// TIA Portal project "TS_Stoliar_DP" (V20)

(* hardware
DEVICE "S7-1200 G2 station_1"  S7-1200 G2 Station
   slot 0: "Rack_0"  S71200G2 Rack  Rack  V1.0
   slot 1: "G2_PLC_1"  CPU 1214C DC/DC/DC  6ES7 214-1AH50-0XB0  V1.0
   slot 9: "AI2/AQ2 signal board_1"  AI2/AQ2 signal board  6ES7 233-4HD50-0XB0  V1.0
*)

// ===== PLC "G2_PLC_1"  CPU 1214C DC/DC/DC =====

VAR_GLOBAL   // PLC tag table "Default tag table"
   "VENT" AT %QW80 : Int;
   "SPIR" AT %QW82 : Int;
   "SNIMAC1" AT %IW80 : Int;
   "SNIMAC2" AT %IW82 : Int;
END_VAR

DATA_BLOCK "DATA"   // DB1
{ S7_Optimized_Access := 'TRUE' }
VERSION : 0.1
   VAR
      block_enable : Bool;
      y1 : Real;
      y2 : Real;
      u : Real;
      vent : Real;
      "time" : LReal;
      ypb : Real;
      u_pb : Real;
   END_VAR
BEGIN
END_DATA_BLOCK

DATA_BLOCK "Current_time_DB"   // DB2
{ S7_Optimized_Access := 'TRUE' }
VERSION : 0.1
// stored: InstanceOfName Current_time
"Current_time"
BEGIN
END_DATA_BLOCK

DATA_BLOCK "PREP"   // DB3
{ S7_Optimized_Access := 'TRUE' }
VERSION : 0.1
   VAR
      r_l : Real;
      r_g : Real;
      r_gf : Real;
      u_g : Real;
      u_l : Real;
      active_g : Bool;
      Ki_l : Real;
      Kp_l : Real;
   END_VAR
BEGIN
END_DATA_BLOCK

DATA_BLOCK "FB_PI_TS05_DB"   // DB5
{ S7_Optimized_Access := 'TRUE' }
VERSION : 0.1
// stored: InstanceOfName FB_PI_TS05
"FB_PI_TS05"
BEGIN
END_DATA_BLOCK

DATA_BLOCK "FB_PI_LOGGER_DB"   // DB6
{ S7_Optimized_Access := 'TRUE' }
VERSION : 0.1
// stored: InstanceOfName FB_PI_LOGGER
"FB_PI_LOGGER"
BEGIN
END_DATA_BLOCK

// folder: System blocks/Program resources

DATA_BLOCK "IEC_Timer_0_DB"   // DB4
{ S7_Optimized_Access := 'TRUE' }
AUTHOR : Simatic
FAMILY : IEC
NAME : IEC_TMR
VERSION : 1.0
// stored: InstanceOfName IEC_TIMER
"IEC_TIMER"
BEGIN
END_DATA_BLOCK

// folder: (top level)

FUNCTION_BLOCK "FB_PI_TS05"   // FB1, SCL
{ S7_Optimized_Access := 'TRUE' }
VERSION : 0.1
   VAR_INPUT
      Y : Real;
      Setpoint_pb : Real;
      Enable : Bool;
   END_VAR
   VAR_OUTPUT
      U : Real;
      Ypb : Real;
      vent : Real;
   END_VAR
   VAR
      Integrator : Real;
   END_VAR
   VAR_TEMP
      "E" : Real;
      DU : Real;
   END_VAR
   VAR CONSTANT
      Kp : Real := 3.58;
      Ki : Real := 1.84;
      Ts : Real := 0.1;
      U_pb : Real := 4.0;
      DU_min : Real := -4.0;
      DU_max : Real := 6.0;
   END_VAR
BEGIN
   IF NOT #Enable THEN
       #U := #U_pb;
       #DU := 0.0;
       #E := 0.0;
       #Integrator := 0.0;
       #Ypb := #Y;
       #vent := 6.0;

   ELSE
       #E := #Setpoint_pb - (#Y - #Ypb);
       #Integrator := #Integrator + #E * #Ts;

       #DU := #Kp * #E + #Ki * #Integrator;

       IF #DU > #DU_max THEN
           #DU := #DU_max;
       ELSIF #DU < #DU_min THEN
           #DU := #DU_min;
       END_IF;

       #U := #U_pb + #DU;
       #vent := 6.0;
   END_IF;
END_FUNCTION_BLOCK

FUNCTION_BLOCK "FB_PI_LOGGER"   // FB2, SCL
{ S7_Optimized_Access := 'TRUE' }
VERSION : 0.1
   VAR_INPUT
      CurrentTimeSec : LReal;
      u : Real;
      y : Real;
      r : Real;
      ypb : Real;
      Enable : Bool;
   END_VAR
   VAR_OUTPUT
      SampleCount : DInt;
      Full : Bool;
   END_VAR
   VAR
      idx : DInt;
      TimeLog_s : Array[0..9999] of LReal;
      ULOG : Array[0..9999] of Real;
      YLOG : Array[0..9999] of Real;
      RLOG : Array[0..9999] of Real;
      YPBLOG : Array[0..9999] of Real;
   END_VAR
BEGIN
   IF NOT #Full AND #Enable THEN
       IF #idx <= 9999 THEN
           #TimeLog_s[#idx] := #CurrentTimeSec;
           #ULOG[#idx] := #u;
           #YLOG[#idx] := #y;
           #RLOG[#idx] := #r;
           #YPBLOG[#idx] := #ypb;

           #idx := #idx + 1;
           #SampleCount := #idx;
       ELSE
           #Full := TRUE;
       END_IF;
   END_IF;
END_FUNCTION_BLOCK

FUNCTION_BLOCK "Current_time"   // FB3, SCL
{ S7_Optimized_Access := 'TRUE' }
VERSION : 0.1
   VAR_OUTPUT
      CurrentTimeSec : LReal;
   END_VAR
   VAR
      started : Bool;
      retVal : Int;
      startTime : DTL;
      currentTime : DTL;
      elapsedTime : Time;
   END_VAR
BEGIN
   #retVal := RD_SYS_T(OUT => #currentTime);

   IF (NOT #started) AND (#retVal = 0) THEN
       #startTime := #currentTime;
       #started := TRUE;
   END_IF;

   IF #started AND (#retVal = 0) THEN
       #elapsedTime := T_DIFF(IN1 := #currentTime, IN2 := #startTime);
       #CurrentTimeSec := DINT_TO_LREAL(TIME_TO_DINT(#elapsedTime)) / 1000.0;
   ELSE
       #CurrentTimeSec := 0.0;
   END_IF;
END_FUNCTION_BLOCK

FUNCTION_BLOCK "FB_PREP_TS05"   // FB4, SCL
{ S7_Optimized_Access := 'TRUE' }
VERSION : 0.1
   VAR_INPUT
      Y : Real;
      R_g : Real;
      R_l : Real;
      Enable : Bool;
      Vent_in : Real;
   END_VAR
   VAR_OUTPUT
      U : Real;
      R_gf : Real;
      Y_pb_out : Real;
      U_pb_out : Real;
      U_g : Real;
      U_l : Real;
      Active_g : Bool;
      Kp_l_out : Real;
      Ki_l_out : Real;
      Vent_out : Real;
   END_VAR
   VAR
      X_f1 : Real;
      X_f2 : Real;
      I_l : Real;
      I_g : Real;
      Y_hist : Array[0..29] of Real;
      U_hist : Array[0..29] of Real;
      R_g_prev : Real;
      Active_g_m : Bool;
      Y_pb : Real;
      U_pb : Real;
      Initialized : Bool;
      Y_pb_table : Array[0..2] of Real;
      U_pb_table : Array[0..2] of Real;
      Kp_l_table : Array[0..2] of Real;
      Ki_l_table : Array[0..2] of Real;
   END_VAR
   VAR_TEMP
      E_l : Real;
      E_g : Real;
      U_tmp : Real;
      Lower_bound : Real;
      Upper_bound : Real;
      Y_pb_new : Real;
      U_pb_new : Real;
      Count_ok : Int;
      Idx_pb : Int;
      I : Int;
      Active_g_new : Bool;
      Active_l : Bool;
      Kp_l : Real;
      Ki_l : Real;
      Y_pb_est : Real;
      U_pb_est : Real;
      Dist_pb : Real;
      Dist_i : Real;
      X_f1_new : Real;
      X_f2_new : Real;
      Mean_y : Real;
      Mean_u : Real;
   END_VAR
   VAR CONSTANT
      Ts : Real := 0.1;
      Kp_g : Real := 4.0;
      Ki_g : Real := 0.7;
   END_VAR
BEGIN
   IF NOT #Enable THEN
       #U := 0.0;
       #R_gf := 0.0;
       #Y_pb_out := #Y_pb;
       #U_pb_out := #U_pb;
       #U_g := 0.0;
       #U_l := 0.0;
       #Active_g := #Active_g_m;
       #Kp_l_out := 0.0;
       #Ki_l_out := 0.0;
       #Vent_out := #Vent_in;
       RETURN;
   END_IF;

   // One-time initialization
   IF NOT #Initialized THEN
       #X_f1 := 0.0;
       #X_f2 := 0.0;
       #I_l := 0.0;
       #I_g := 0.0;
       #R_g_prev := #R_g;
       #Active_g_m := FALSE;
       #Y_pb := 0.0;
       #U_pb := 0.0;

       #Y_pb_table[0] := 4.4884;
       #Y_pb_table[1] := 6.3412;
       #Y_pb_table[2] := 7.7441;

       #U_pb_table[0] := 2.0;
       #U_pb_table[1] := 4.0;
       #U_pb_table[2] := 6.0;

       #Kp_l_table[0] := 2.77;
       #Kp_l_table[1] := 3.58;
       #Kp_l_table[2] := 1.83;

       #Ki_l_table[0] := 1.48;
       #Ki_l_table[1] := 1.84;
       #Ki_l_table[2] := 2.20;

       FOR #I := 0 TO 29 DO
           #Y_hist[#I] := 0.0;
           #U_hist[#I] := 0.0;
       END_FOR;

       #Initialized := TRUE;
   END_IF;

   // 1 Detect step change of global reference
   IF #R_g <> #R_g_prev THEN
       #Active_g_m := TRUE;
   END_IF;

   // 2 Filter global reference
   #R_gf := 0.01 * #X_f1;

   #X_f1_new := #X_f1 + #Ts * #X_f2;
   #X_f2_new := #X_f2 + #Ts * (-0.01 * #X_f1 - 0.2 * #X_f2 + #R_g);

   // 3 Select local operating point and PI parameters from table
   #Dist_pb := ABS(#Y_pb_table[0] - #Y_pb);
   #Idx_pb := 0;

   FOR #I := 1 TO 2 DO
       #Dist_i := ABS(#Y_pb_table[#I] - #Y_pb);
       IF #Dist_i < #Dist_pb THEN
           #Dist_pb := #Dist_i;
           #Idx_pb := #I;
       END_IF;
   END_FOR;

   #Kp_l := #Kp_l_table[#Idx_pb];
   #Ki_l := #Ki_l_table[#Idx_pb];

   // 4 Control errors
   #E_l := #R_l - (#Y - #Y_pb);
   #E_g := #R_gf - #Y;

   // 5 Control law
   IF #Active_g_m THEN
       #U_l := 0.0;
       #U_g := #Kp_g * #E_g + #Ki_g * #I_g;
   ELSE
       #U_l := #U_pb + #Kp_l * #E_l + #Ki_l * #I_l;
       #U_g := 0.0;
   END_IF;

   #U_tmp := #U_l + #U_g;

   // Saturation
   IF #U_tmp > 10.0 THEN
       #U_tmp := 10.0;
   ELSIF #U_tmp < 0.0 THEN
       #U_tmp := 0.0;
   END_IF;

   #U := #U_tmp;

   // 6 Update histories
   FOR #I := 0 TO 28 DO
       #Y_hist[#I] := #Y_hist[#I + 1];
       #U_hist[#I] := #U_hist[#I + 1];
   END_FOR;

   #Y_hist[29] := #Y;
   #U_hist[29] := #U;

   // 7 Settling detection
   #Lower_bound := #R_g - 0.03 * #R_g;
   #Upper_bound := #R_g + 0.03 * #R_g;

   #Count_ok := 0;
   FOR #I := 0 TO 29 DO
       IF (#Y_hist[#I] >= #Lower_bound) AND (#Y_hist[#I] <= #Upper_bound) THEN
           #Count_ok := #Count_ok + 1;
       END_IF;
   END_FOR;

   // Two-level switching logic
   #Y_pb_new := #Y_pb;
   #U_pb_new := #U_pb;
   #Active_g_new := #Active_g_m;

   IF #Active_g_m AND (#Count_ok >= 25) THEN
       #Mean_y := 0.0;
       #Mean_u := 0.0;

       FOR #I := 0 TO 29 DO
           #Mean_y := #Mean_y + #Y_hist[#I];
           #Mean_u := #Mean_u + #U_hist[#I];
       END_FOR;

       #Y_pb_est := #Mean_y / 30.0;
       #U_pb_est := #Mean_u / 30.0;

       #Y_pb_new := #Y_pb_est;
       #U_pb_new := #U_pb_est;
       #Active_g_new := FALSE;
   END_IF;

   IF #Active_g_m THEN
       #Active_l := FALSE;
   ELSE
       #Active_l := TRUE;
   END_IF;

   // 8 Integral states update
   IF #Active_l THEN
       #I_l := #I_l + #E_l * #Ts;
   ELSE
       #I_l := 0.0;
   END_IF;

   IF #Active_g_m THEN
       #I_g := #I_g + #E_g * #Ts;
   ELSE
       #I_g := (#U - #Kp_g * #E_g) / #Ki_g;
   END_IF;

   // 9 Memory update
   #R_g_prev := #R_g;
   #Y_pb := #Y_pb_new;
   #U_pb := #U_pb_new;
   #Active_g_m := #Active_g_new;
   #X_f1 := #X_f1_new;
   #X_f2 := #X_f2_new;

   // Outputs for monitoring/logging
   #Y_pb_out := #Y_pb;
   #U_pb_out := #U_pb;
   #Active_g := #Active_g_m;
   #Kp_l_out := #Kp_l;
   #Ki_l_out := #Ki_l;
   #Vent_out := #Vent_in;
END_FUNCTION_BLOCK

FUNCTION_BLOCK "FB_PREP_LOGGER"   // FB5, SCL
{ S7_Optimized_Access := 'TRUE' }
VERSION : 0.1
   VAR_INPUT
      t : LReal;
      r_l : Real;
      r_g : Real;
      r_gf : Real;
      y : Real;
      y_pb : Real;
      u : Real;
      u_g : Real;
      u_l : Real;
      u_pb : Real;
      active_g : Bool;
      Ki_l : Real;
      Kp_l : Real;
      Vent : Real;
   END_VAR
   VAR_OUTPUT
      SampleCount : DInt;
      Full : Bool;
   END_VAR
   VAR
      idx : DInt;
      TimeLog_s : Array[0..9999] of LReal;
      R_L_log : Array[0..9999] of Real;
      R_G_log : Array[0..9999] of Real;
      R_GF_log : Array[0..9999] of Real;
      Y_log : Array[0..9999] of Real;
      Y_PB_log : Array[0..9999] of Real;
      U_log : Array[0..9999] of Real;
      U_G_log : Array[0..9999] of Real;
      U_L_log : Array[0..9999] of Real;
      U_PB_log : Array[0..9999] of Real;
      ACTIVE_G_log : Array[0..9999] of Bool;
      KI_L_log : Array[0..9999] of Real;
      KP_L_log : Array[0..9999] of Real;
      VENT_log : Array[0..9999] of Real;
   END_VAR
BEGIN
   IF NOT #Full THEN
       IF #idx <= 9999 THEN
           #TimeLog_s[#idx] := #t;
           #R_L_log[#idx] := #r_l;
           #R_G_log[#idx] := #r_g;
           #R_GF_log[#idx] := #r_gf;
           #Y_log[#idx] := #y;
           #Y_PB_log[#idx] := #y_pb;
           #U_log[#idx] := #u;
           #U_G_log[#idx] := #u_g;
           #U_L_log[#idx] := #u_l;
           #U_PB_log[#idx] := #u_pb;
           #ACTIVE_G_log[#idx] := #active_g;
           #KI_L_log[#idx] := #Ki_l;
           #KP_L_log[#idx] := #Kp_l;
           #VENT_log[#idx] := #Vent;

           #idx := #idx + 1;
           #SampleCount := #idx;
       ELSE
           #Full := TRUE;
       END_IF;
   END_IF;
END_FUNCTION_BLOCK

FUNCTION_BLOCK "FB_PREP_SETPOINT"   // FB6, SCL
{ S7_Optimized_Access := 'TRUE' }
VERSION : 0.1
   VAR_INPUT
      t : LReal;
   END_VAR
   VAR_OUTPUT
      r_l : Real;
      r_g : Real;
   END_VAR
BEGIN
   IF #t < 1.0 THEN
       #r_g := 0.0;
   ELSIF #t < 401.0 THEN
       #r_g := 6.3412;
   ELSIF #t < 801.0 THEN
       #r_g := 4.4884;
   ELSE
       #r_g := 4.4884;
   END_IF;

   IF #t < 201.0 THEN
       #r_l := 0.0;
   ELSIF #t < 301.0 THEN
       #r_l := -0.35;
   ELSIF #t < 601.0 THEN
       #r_l := 0.0;
   ELSIF #t < 701.0 THEN
       #r_l := 0.41;
   ELSIF #t < 801.0 THEN
       #r_l := 0.0;
   ELSE
       #r_l := 0.0;
   END_IF;
END_FUNCTION_BLOCK

ORGANIZATION_BLOCK "Main"   // OB1, LAD, ProgramCycle
TITLE = "Main Program Sweep (Cycle)"
{ S7_Optimized_Access := 'TRUE' }
VERSION : 0.1
   VAR_INPUT
      Initial_Call : Bool;   // Initial call of this OB
      Remanence : Bool;   // =True, if remanent data are available
   END_VAR
   VAR_TEMP
      temp_real : Real;
   END_VAR
BEGIN

REGION Network 1
   // Time counting
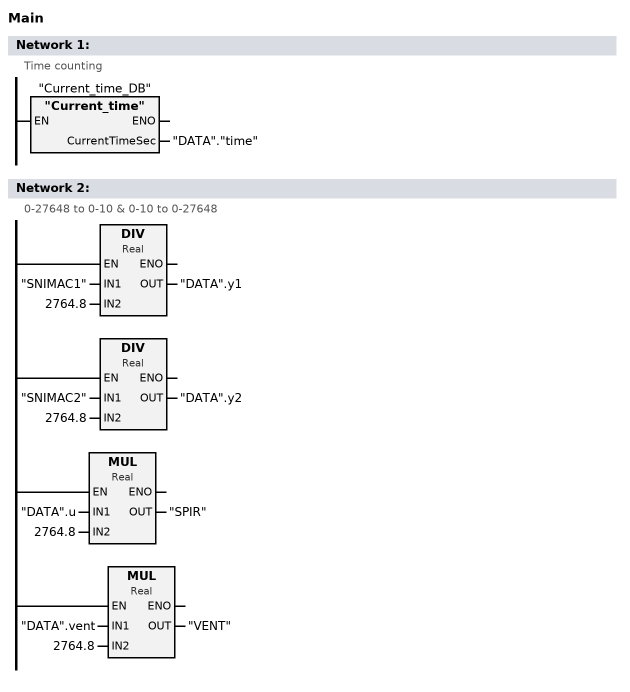
   RUNG wire#powerrail
      "Current_time_DB"(CurrentTimeSec => "DATA"."time")
   END_RUNG
   // the same network as SCL:
   "Current_time_DB"(CurrentTimeSec => "DATA"."time");   // "Current_time"
END_REGION

REGION Network 2
   // 0-27648 to 0-10 & 0-10 to 0-27648
   RUNG wire#powerrail
      { S7_Templates := "SrcType := Real" } Div(in1 := "SNIMAC1", in2 := 2764.8, out => "DATA".y1)
   END_RUNG
   RUNG wire#powerrail
      { S7_Templates := "SrcType := Real" } Div(in1 := "SNIMAC2", in2 := 2764.8, out => "DATA".y2)
   END_RUNG
   RUNG wire#powerrail
      { S7_Templates := "SrcType := Real" } Mul(in1 := "DATA".u, in2 := 2764.8, out => "SPIR")
   END_RUNG
   RUNG wire#powerrail
      { S7_Templates := "SrcType := Real" } Mul(in1 := "DATA".vent, in2 := 2764.8, out => "VENT")
   END_RUNG
   // the same network as SCL:
   "DATA".y1 := "SNIMAC1" / 2764.8;
   "DATA".y2 := "SNIMAC2" / 2764.8;
   "SPIR" := "DATA".u * 2764.8;
   "VENT" := "DATA".vent * 2764.8;
END_REGION
END_ORGANIZATION_BLOCK

ORGANIZATION_BLOCK "CyclicInterrupt"   // OB30, LAD, CyclicInterrupt
{ S7_Optimized_Access := 'TRUE' }
VERSION : 0.1
   VAR_INPUT
      Initial_Call : Bool;   // Initial call of this OB
      Event_Count : Int;   // Events discarded
   END_VAR
   VAR_TEMP   // added for the SCL form of the ladder/FBD networks
      _w1 : Bool;
   END_VAR
BEGIN

REGION Network 1
   // CONTROL LOGIC
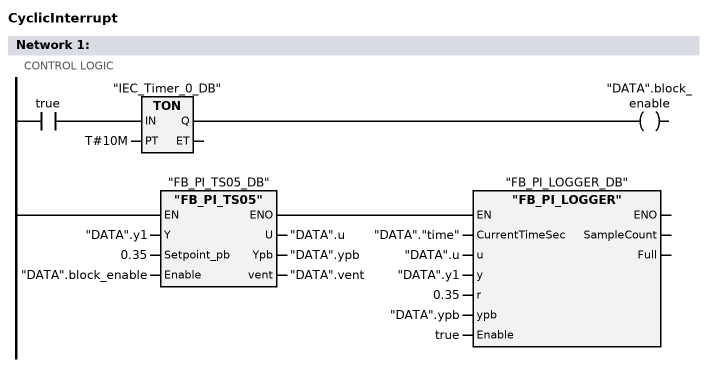
   "IEC_Timer_0_DB".TON(IN := true, PT := T#10M);
   "DATA".block_enable := "IEC_Timer_0_DB".Q;
   "FB_PI_TS05_DB"(Y := "DATA".y1,   // "FB_PI_TS05"
                   Setpoint_pb := 0.35,
                   Enable := "DATA".block_enable,
                   U => "DATA".u,
                   Ypb => "DATA".ypb,
                   vent => "DATA".vent,
                   ENO => #_w1);
   IF #_w1 THEN
       "FB_PI_LOGGER_DB"(CurrentTimeSec := "DATA"."time",   // "FB_PI_LOGGER"
                         u := "DATA".u,
                         y := "DATA".y1,
                         r := 0.35,
                         ypb := "DATA".ypb,
                         Enable := true);
   END_IF;
END_REGION
END_ORGANIZATION_BLOCK